{attribute 'call_after_init'}
FUNCTION_BLOCK FB_GantryAutoCoupling_Test EXTENDS TcUnit.FB_TestSuite

CoupledOnStartup();

METHOD PRIVATE CoupledOnStartup
VAR_INST
	fbAutoCouple : FB_GantryAutoCoupling;

	// @TEST-FIXTURE EmergencyErrorCode
	fbMotionStage_M1, fbMotionStage_M2 : FB_MotionStage;

	nCycleCount : ULINT := 0;
END_VAR
VAR
	bStartCouple : BOOL;
	bStopCouple : BOOL;

	// @TEST-RESULT CouplingStatus
	ExpectedStatus : BOOL := TRUE;
	WatchCouplingStatus : BOOL;
	CouplingStatus : BOOL;
END_VAR
TEST('CoupledOnStartup');

nCycleCount := nCycleCount + 1;

TestAxes.M1.bGantryAxis := TRUE;
TestAxes.M1.fGantryTol := 50000;
TestAxes.M1.nCommand := 3;
TestAxes.M2.bGantryAxis := TRUE;
TestAxes.M2.fGantryTol := TestAxes.M1.fGantryTol;

TestAxes.master_enc.Count := LREAL_TO_ULINT(TestAxes.M1.stAxisStatus.fActPosition * EXPT(10, 6));
TestAxes.slave_enc.Count := LREAL_TO_ULINT(TestAxes.M1.stAxisStatus.fActPosition * EXPT(10, 6));

// @TEST-RUN
fbMotionStage_M1(stMotionStage:=TestAxes.M1);
fbMotionStage_M2(stMotionStage:=TestAxes.M2);

WatchCouplingStatus := TestAxes.M1.Axis.NcToPlc.CoupleState=1 AND TestAxes.M2.Axis.NcToPlc.CoupleState=3;



fbAutoCouple(fGantryTol:=5000, Master:=TestAxes.M1, MasterEnc:=TestAxes.master_enc, Slave:=TestAxes.M2,
	         SlaveEnc:=TestAxes.slave_enc, bExecuteCouple:=bStartCouple,
			 bExecuteDecouple:=bStopCouple,
			 bGantryAlreadyCoupled=>CouplingStatus);

IF nCycleCount = 2 THEN
	// @TEST-ASSERT
	AssertEquals(Expected:=ExpectedStatus, Actual:=CouplingStatus,
	         	 Message:='Master and Slave did not start coupled');

	TEST_FINISHED('');
END_IF
END_METHOD

END_FUNCTION_BLOCK

(* stored: Version 1.1.0.1, ProductVersion 3.1.4022.12
   POU FB_GantryAutoCoupling_Test: Id {3e5c3561-28ef-436b-b33a-73b0af1b1acd}, SpecialFunc None
   Method CoupledOnStartup: Id {14e0e036-d1c6-49ab-8e38-ef361b3960ec} *)
